// Minimal I_Comm stub for tests: every Publish/PublishLog call is a no-op that reports success,
// so FBs under test can call fbComm.Publish(...) freely without a real MQTT connection.
FUNCTION_BLOCK FB_NullComm IMPLEMENTS BROTLib.I_Comm
VAR
END_VAR

METHOD Publish : BOOL
VAR_INPUT
	domain			: STRING(255) := 'environment';
	location		: STRING(255) := 'roof';
	parameter		: STRING(255);
	value			: STRING(255);
END_VAR
VAR_OUTPUT
	published	: BOOL;
END_VAR
Publish := TRUE;
published := TRUE;
END_METHOD

METHOD PublishLog : BOOL
VAR_INPUT
	level		: STRING(255) := 'INFO';
	message		: STRING(255);
END_VAR
VAR_OUTPUT
	published	: BOOL;
END_VAR
PublishLog := TRUE;
published := TRUE;
END_METHOD

END_FUNCTION_BLOCK

(* stored: Version 1.1.0.1, ProductVersion 3.1.4024.15
   POU FB_NullComm: Id {733d720e-0516-4a55-a5a5-f72ebf9f58f9}, SpecialFunc None
   Method Publish: Id {79b3e026-bcb6-4a3a-bdc7-e228b153f1bc}
   Method PublishLog: Id {27dc438e-e3f1-4f55-b4bb-810991230d3e} *)
